{attribute 'GeneratedUsingTerminal: AT2025-0250-0023'}
{attribute addProperty BoxType "AT2025-0250-0023"}
{attribute addProperty Id "A_0076_AT2001_5250_0017_AT2001_5250AT2001_33A3DF1B80"}
{attribute addProperty CRC "2303684572"}
{attribute addProperty Size "80"}
TYPE A_0064_AT2025_0250_0023_AT2025_0250_894F6FDC EXTENDS AT2025_2EA6C9BF :
STRUCT
	{attribute addProperty Name "A_0076(AT2001-5250-0017) (AT2001-5250)"}
	{attribute addProperty PreviousPort "A_0064(AT2025-0250-0023) (AT2025-0250) : B"}
	A_0076_AT2001_5250_0017_AT2001_5250 : AT2001_33A3DF1B;
END_STRUCT
END_TYPE

(* stored: Version 1.2.0.0, ProductVersion 3.1.4024.9
   DUT A_0064_AT2025_0250_0023_AT2025_0250_894F6FDC: Id {d55b6814-3ab9-4734-b80d-c477a0003310} *)
